{attribute 'linkalways'} 
{attribute 'no_explicit_call' := 'This FB is a CLASS and must be accessed using methods or properties'}
{attribute 'enable_dynamic_creation'}
FUNCTION_BLOCK Node_F_VN_InsertIntoContainer_TcVnVector4_LREAL EXTENDS VisionNode
VAR
    aElement : _TcVnVector4_LREAL;
    ipContainer : _ITcVnContainer;
    nIndex : _ULINT(0);
    hrPrev : _HRESULT(S_OK);
    hresult : _HRESULT(S_OK);
END_VAR

METHOD PUBLIC  Clone : I_Node
VAR
	pNode : POINTER TO Node_F_VN_InsertIntoContainer_TcVnVector4_LREAL;
END_VAR
pNode := __NEW(Node_F_VN_InsertIntoContainer_TcVnVector4_LREAL);
Clone := pNode^;
END_METHOD

METHOD FB_init : BOOL
VAR_INPUT
	bInitRetains : BOOL; // if TRUE, the retain variables are initialized (warm start / cold start)
	bInCopyCode : BOOL;  // if TRUE, the instance afterwards gets moved into the copy code (online change)
END_VAR
AddInput('aElement', aElement);
AddInput('ipContainer', ipContainer);
AddInput('nIndex', nIndex);
AddInput('hrPrev', hrPrev);
AddOutput('ipContainer', ipContainer);
AddOutput('hresult',hresult);
END_METHOD

METHOD PROTECTED OnExecute : HRESULT
hresult.Value := F_VN_InsertIntoContainer_TcVnVector4_LREAL(
    aElement := aElement.Value,
    ipContainer := ipContainer.Value,
    nIndex := nIndex.Value,
    hrPrev:= hrPrev.Value);
END_METHOD

METHOD PUBLIC PreExecutionCheck
VAR_INPUT
	Check : I_PreExecutionChecks;
END_VAR
Check.IsTrue(ipContainer.IsValid, 'ipContainer must be a valid container');
END_METHOD

END_FUNCTION_BLOCK

(* stored: Version 1.1.0.1, ProductVersion 3.1.4024.13
   POU Node_F_VN_InsertIntoContainer_TcVnVector4_LREAL: Id {9ecf173d-d056-47e7-8b60-424bd9a1a6b6}, SpecialFunc None
   Folder Constructor: Id {2acd8e1f-9998-450c-acbb-1ff70580671f}
   Method Clone: Id {88d5d5c3-213a-4421-9ba7-923479b7604b}
   Method FB_init: Id {7c80cd99-750e-42bd-b2b7-1ad590ef052d}
   Method OnExecute: Id {b3ef4c9d-f5a4-47fc-a425-c0035911c13c}
   Method PreExecutionCheck: Id {0987051c-93e9-4fee-8f5b-aba5cf738d4d} *)
